MDP5001_342_DPM_Variant_Value_Out_Index_1_REAL_1	:= 		prgEM.stEL3446_IO_1.MDP5001_342_Output.MDP5001_342_DPM_Variant_Value_Out_Index_1_REAL	;
MDP5001_342_DPM_Variant_Value_Out_Index_2_REAL_1	:= 		prgEM.stEL3446_IO_1.MDP5001_342_Output.MDP5001_342_DPM_Variant_Value_Out_Index_2_REAL	;	
MDP5001_342_DPM_Variant_Value_Out_Index_3_REAL_1	:= 		prgEM.stEL3446_IO_1.MDP5001_342_Output.MDP5001_342_DPM_Variant_Value_Out_Index_3_REAL	;
MDP5001_342_DPM_Variant_Value_Out_Index_4_ULINT_1	:= 		prgEM.stEL3446_IO_1.MDP5001_342_Output.MDP5001_342_DPM_Variant_Value_Out_Index_4_ULINT	;
MDP5001_342_DPM_Data_Data_1_1						:= 		prgEM.stEL3446_IO_1.MDP5001_342_Output.MDP5001_342_DPM_Data_Data_1	;
MDP5001_342_DPM_Data_Data_2_1						:= 		prgEM.stEL3446_IO_1.MDP5001_342_Output.MDP5001_342_DPM_Data_Data_2	;
MDP5001_342_DPM_Data_Data_3_1						:= 		prgEM.stEL3446_IO_1.MDP5001_342_Output.MDP5001_342_DPM_Data_Data_3	;
MDP5001_342_DPM_Data_Data_4_1						:= 		prgEM.stEL3446_IO_1.MDP5001_342_Output.MDP5001_342_DPM_Data_Data_4	;
MDP5001_342_DPM_Data_Data_5_1						:= 		prgEM.stEL3446_IO_1.MDP5001_342_Output.MDP5001_342_DPM_Data_Data_5	;
MDP5001_342_DPM_Data_Data_6_1						:= 		prgEM.stEL3446_IO_1.MDP5001_342_Output.MDP5001_342_DPM_Data_Data_6	;
MDP5001_342_DPM_Data_Data_7_1						:= 		prgEM.stEL3446_IO_1.MDP5001_342_Output.MDP5001_342_DPM_Data_Data_7	;
MDP5001_342_DPM_Data_Data_8_1						:= 		prgEM.stEL3446_IO_1.MDP5001_342_Output.MDP5001_342_DPM_Data_Data_8	;
MDP5001_342_DPM_Data_Data_9_1						:= 		prgEM.stEL3446_IO_1.MDP5001_342_Output.MDP5001_342_DPM_Data_Data_9	;
MDP5001_342_DPM_Data_Data_10_1						:= 		prgEM.stEL3446_IO_1.MDP5001_342_Output.MDP5001_342_DPM_Data_Data_10	;
MDP5001_342_DPM_Data_Data_11_1						:= 		prgEM.stEL3446_IO_1.MDP5001_342_Output.MDP5001_342_DPM_Data_Data_11	;
MDP5001_342_DPM_Data_Data_12_1						:= 		prgEM.stEL3446_IO_1.MDP5001_342_Output.MDP5001_342_DPM_Data_Data_12	;
MDP5001_342_DPM_Data_Data_13_1						:= 		prgEM.stEL3446_IO_1.MDP5001_342_Output.MDP5001_342_DPM_Data_Data_13	;
MDP5001_342_DPM_Data_Data_14_1						:= 		prgEM.stEL3446_IO_1.MDP5001_342_Output.MDP5001_342_DPM_Data_Data_14	;
MDP5001_342_DPM_Data_Data_15_1						:= 		prgEM.stEL3446_IO_1.MDP5001_342_Output.MDP5001_342_DPM_Data_Data_15	;
MDP5001_342_DPM_Data_Data_16_1						:= 		prgEM.stEL3446_IO_1.MDP5001_342_Output.MDP5001_342_DPM_Data_Data_16	;
MDP5001_342_DPM_Data_Data_17_1						:= 		prgEM.stEL3446_IO_1.MDP5001_342_Output.MDP5001_342_DPM_Data_Data_17	;
MDP5001_342_DPM_Data_Data_18_1						:= 		prgEM.stEL3446_IO_1.MDP5001_342_Output.MDP5001_342_DPM_Data_Data_18	;
MDP5001_342_DPM_Data_Data_19_1						:= 		prgEM.stEL3446_IO_1.MDP5001_342_Output.MDP5001_342_DPM_Data_Data_19	;
MDP5001_342_DPM_Data_Data_20_1						:= 		prgEM.stEL3446_IO_1.MDP5001_342_Output.MDP5001_342_DPM_Data_Data_20	;




prgEM.stEL3446_IO_2.MDP5001_342_Input.MDP5001_342_I1_Channel_Overcurrent					:=	MDP5001_342_I1_Channel_Overcurrent_2;
prgEM.stEL3446_IO_2.MDP5001_342_Input.MDP5001_342_I1_Channel_Inaccurate_Current			:=	MDP5001_342_I1_Channel_Inaccurate_Current_2;
prgEM.stEL3446_IO_2.MDP5001_342_Input.MDP5001_342_I1_Channel_Current_Guard_Warning		:=	MDP5001_342_I1_Channel_Current_Guard_Warning_2;
prgEM.stEL3446_IO_2.MDP5001_342_Input.MDP5001_342_I1_Channel_Current_Guard_Error			:=	MDP5001_342_I1_Channel_Current_Guard_Error_2;
prgEM.stEL3446_IO_2.MDP5001_342_Input.MDP5001_342_I1_Channel_Apparent_Power_Guard_Warning	:=	MDP5001_342_I1_Channel_Apparent_Power_Guard_Warning_2;
prgEM.stEL3446_IO_2.MDP5001_342_Input.MDP5001_342_I1_Channel_Apparent_Power_Guard_Error	:=	MDP5001_342_I1_Channel_Apparent_Power_Guard_Error_2;
prgEM.stEL3446_IO_2.MDP5001_342_Input.MDP5001_342_I1_Channel_Active_Power_Guard_Warning	:=	MDP5001_342_I1_Channel_Active_Power_Guard_Warning_2;
prgEM.stEL3446_IO_2.MDP5001_342_Input.MDP5001_342_I1_Channel_Active_Power_Guard_Error		:=	MDP5001_342_I1_Channel_Active_Power_Guard_Error_2;
prgEM.stEL3446_IO_2.MDP5001_342_Input.MDP5001_342_I1_Channel_Reactive_Power_Guard_Warning	:=	MDP5001_342_I1_Channel_Reactive_Power_Guard_Warning_2;
prgEM.stEL3446_IO_2.MDP5001_342_Input.MDP5001_342_I1_Channel_Reactive_Power_Guard_Error	:=	MDP5001_342_I1_Channel_Reactive_Power_Guard_Error_2;
prgEM.stEL3446_IO_2.MDP5001_342_Input.MDP5001_342_I1_Channel_DPM_Inaccurate				:=	MDP5001_342_I1_Channel_DPM_Inaccurate_2;
prgEM.stEL3446_IO_2.MDP5001_342_Input.MDP5001_342_I1_Channel_DPM_Timeout					:=	MDP5001_342_I1_Channel_DPM_Timeout_2;
prgEM.stEL3446_IO_2.MDP5001_342_Input.MDP5001_342_I1_Channel_TxPDO_Toggle					:=	MDP5001_342_I1_Channel_TxPDO_Toggle_2;
prgEM.stEL3446_IO_2.MDP5001_342_Input.MDP5001_342_I1_Channel_Current						:=	MDP5001_342_I1_Channel_Current_2;
prgEM.stEL3446_IO_2.MDP5001_342_Input.MDP5001_342_I1_Channel_Active_Power					:=	MDP5001_342_I1_Channel_Active_Power_2;
prgEM.stEL3446_IO_2.MDP5001_342_Input.MDP5001_342_I1_Channel_Apparent_Power				:=	MDP5001_342_I1_Channel_Apparent_Power_2;
prgEM.stEL3446_IO_2.MDP5001_342_Input.MDP5001_342_I1_Channel_Reactive_Power_Fundamental	:=	MDP5001_342_I1_Channel_Reactive_Power_Fundamental_2;
prgEM.stEL3446_IO_2.MDP5001_342_Input.MDP5001_342_I1_Channel_Active_Energy				:=	MDP5001_342_I1_Channel_Active_Energy_2;
prgEM.stEL3446_IO_2.MDP5001_342_Input.MDP5001_342_I2_Channel_Overcurrent					:=	MDP5001_342_I2_Channel_Overcurrent_2;
prgEM.stEL3446_IO_2.MDP5001_342_Input.MDP5001_342_I2_Channel_Inaccurate_Current			:=	MDP5001_342_I2_Channel_Inaccurate_Current_2;
prgEM.stEL3446_IO_2.MDP5001_342_Input.MDP5001_342_I2_Channel_Current_Guard_Warning		:=	MDP5001_342_I2_Channel_Current_Guard_Warning_2;
prgEM.stEL3446_IO_2.MDP5001_342_Input.MDP5001_342_I2_Channel_Current_Guard_Error			:=	MDP5001_342_I2_Channel_Current_Guard_Error_2;
prgEM.stEL3446_IO_2.MDP5001_342_Input.MDP5001_342_I2_Channel_Apparent_Power_Guard_Warning	:=	MDP5001_342_I2_Channel_Apparent_Power_Guard_Warning_2;
prgEM.stEL3446_IO_2.MDP5001_342_Input.MDP5001_342_I2_Channel_Apparent_Power_Guard_Error	:=	MDP5001_342_I2_Channel_Apparent_Power_Guard_Error_2;
prgEM.stEL3446_IO_2.MDP5001_342_Input.MDP5001_342_I2_Channel_Active_Power_Guard_Warning	:=	MDP5001_342_I2_Channel_Active_Power_Guard_Warning_2;
prgEM.stEL3446_IO_2.MDP5001_342_Input.MDP5001_342_I2_Channel_Active_Power_Guard_Error		:=	MDP5001_342_I2_Channel_Active_Power_Guard_Error_2;
prgEM.stEL3446_IO_2.MDP5001_342_Input.MDP5001_342_I2_Channel_Reactive_Power_Guard_Warning	:=	MDP5001_342_I2_Channel_Reactive_Power_Guard_Warning_2;
prgEM.stEL3446_IO_2.MDP5001_342_Input.MDP5001_342_I2_Channel_Reactive_Power_Guard_Error	:=	MDP5001_342_I2_Channel_Reactive_Power_Guard_Error_2;
prgEM.stEL3446_IO_2.MDP5001_342_Input.MDP5001_342_I2_Channel_DPM_Inaccurate				:=	MDP5001_342_I2_Channel_DPM_Inaccurate_2;
prgEM.stEL3446_IO_2.MDP5001_342_Input.MDP5001_342_I2_Channel_DPM_Timeout					:=	MDP5001_342_I2_Channel_DPM_Timeout_2;
prgEM.stEL3446_IO_2.MDP5001_342_Input.MDP5001_342_I2_Channel_TxPDO_Toggle					:=	MDP5001_342_I2_Channel_TxPDO_Toggle_2;
prgEM.stEL3446_IO_2.MDP5001_342_Input.MDP5001_342_I2_Channel_Current						:=	MDP5001_342_I2_Channel_Current_2;
prgEM.stEL3446_IO_2.MDP5001_342_Input.MDP5001_342_I2_Channel_Active_Power					:=	MDP5001_342_I2_Channel_Active_Power_2;
prgEM.stEL3446_IO_2.MDP5001_342_Input.MDP5001_342_I2_Channel_Apparent_Power				:=	MDP5001_342_I2_Channel_Apparent_Power_2;
prgEM.stEL3446_IO_2.MDP5001_342_Input.MDP5001_342_I2_Channel_Reactive_Power_Fundamental	:=	MDP5001_342_I2_Channel_Reactive_Power_Fundamental_2;
prgEM.stEL3446_IO_2.MDP5001_342_Input.MDP5001_342_I2_Channel_Active_Energy				:=	MDP5001_342_I2_Channel_Active_Energy_2;
prgEM.stEL3446_IO_2.MDP5001_342_Input.MDP5001_342_I3_Channel_Overcurrent					:=	MDP5001_342_I3_Channel_Overcurrent_2;
prgEM.stEL3446_IO_2.MDP5001_342_Input.MDP5001_342_I3_Channel_Inaccurate_Current			:=	MDP5001_342_I3_Channel_Inaccurate_Current_2;
prgEM.stEL3446_IO_2.MDP5001_342_Input.MDP5001_342_I3_Channel_Current_Guard_Warning		:=	MDP5001_342_I3_Channel_Current_Guard_Warning_2;
prgEM.stEL3446_IO_2.MDP5001_342_Input.MDP5001_342_I3_Channel_Current_Guard_Error			:=	MDP5001_342_I3_Channel_Current_Guard_Error_2;
prgEM.stEL3446_IO_2.MDP5001_342_Input.MDP5001_342_I3_Channel_Apparent_Power_Guard_Warning	:=	MDP5001_342_I3_Channel_Apparent_Power_Guard_Warning_2;
prgEM.stEL3446_IO_2.MDP5001_342_Input.MDP5001_342_I3_Channel_Apparent_Power_Guard_Error	:=	MDP5001_342_I3_Channel_Apparent_Power_Guard_Error_2;
prgEM.stEL3446_IO_2.MDP5001_342_Input.MDP5001_342_I3_Channel_Active_Power_Guard_Warning	:=	MDP5001_342_I3_Channel_Active_Power_Guard_Warning_2;
prgEM.stEL3446_IO_2.MDP5001_342_Input.MDP5001_342_I3_Channel_Active_Power_Guard_Error		:=	MDP5001_342_I3_Channel_Active_Power_Guard_Error_2;
prgEM.stEL3446_IO_2.MDP5001_342_Input.MDP5001_342_I3_Channel_Reactive_Power_Guard_Warning	:=	MDP5001_342_I3_Channel_Reactive_Power_Guard_Warning_2;
prgEM.stEL3446_IO_2.MDP5001_342_Input.MDP5001_342_I3_Channel_Reactive_Power_Guard_Error	:=	MDP5001_342_I3_Channel_Reactive_Power_Guard_Error_2;
prgEM.stEL3446_IO_2.MDP5001_342_Input.MDP5001_342_I3_Channel_DPM_Inaccurate				:=	MDP5001_342_I3_Channel_DPM_Inaccurate_2;
prgEM.stEL3446_IO_2.MDP5001_342_Input.MDP5001_342_I3_Channel_DPM_Timeout					:=	MDP5001_342_I3_Channel_DPM_Timeout_2;
prgEM.stEL3446_IO_2.MDP5001_342_Input.MDP5001_342_I3_Channel_TxPDO_Toggle					:=	MDP5001_342_I3_Channel_TxPDO_Toggle_2;
prgEM.stEL3446_IO_2.MDP5001_342_Input.MDP5001_342_I3_Channel_Current						:=	MDP5001_342_I3_Channel_Current_2;
prgEM.stEL3446_IO_2.MDP5001_342_Input.MDP5001_342_I3_Channel_Active_Power					:=	MDP5001_342_I3_Channel_Active_Power_2;
prgEM.stEL3446_IO_2.MDP5001_342_Input.MDP5001_342_I3_Channel_Apparent_Power				:=	MDP5001_342_I3_Channel_Apparent_Power_2;
prgEM.stEL3446_IO_2.MDP5001_342_Input.MDP5001_342_I3_Channel_Reactive_Power_Fundamental	:=	MDP5001_342_I3_Channel_Reactive_Power_Fundamental_2;
prgEM.stEL3446_IO_2.MDP5001_342_Input.MDP5001_342_I3_Channel_Active_Energy				:=	MDP5001_342_I3_Channel_Active_Energy_2;
prgEM.stEL3446_IO_2.MDP5001_342_Input.MDP5001_342_I4_Channel_Overcurrent					:=	MDP5001_342_I4_Channel_Overcurrent_2;
prgEM.stEL3446_IO_2.MDP5001_342_Input.MDP5001_342_I4_Channel_Inaccurate_Current			:=	MDP5001_342_I4_Channel_Inaccurate_Current_2;
prgEM.stEL3446_IO_2.MDP5001_342_Input.MDP5001_342_I4_Channel_Current_Guard_Warning		:=	MDP5001_342_I4_Channel_Current_Guard_Warning_2;
prgEM.stEL3446_IO_2.MDP5001_342_Input.MDP5001_342_I4_Channel_Current_Guard_Error			:=	MDP5001_342_I4_Channel_Current_Guard_Error_2;
prgEM.stEL3446_IO_2.MDP5001_342_Input.MDP5001_342_I4_Channel_Apparent_Power_Guard_Warning	:=	MDP5001_342_I4_Channel_Apparent_Power_Guard_Warning_2;
prgEM.stEL3446_IO_2.MDP5001_342_Input.MDP5001_342_I4_Channel_Apparent_Power_Guard_Error	:=	MDP5001_342_I4_Channel_Apparent_Power_Guard_Error_2;
prgEM.stEL3446_IO_2.MDP5001_342_Input.MDP5001_342_I4_Channel_Active_Power_Guard_Warning	:=	MDP5001_342_I4_Channel_Active_Power_Guard_Warning_2;
prgEM.stEL3446_IO_2.MDP5001_342_Input.MDP5001_342_I4_Channel_Active_Power_Guard_Error		:=	MDP5001_342_I4_Channel_Active_Power_Guard_Error_2;
prgEM.stEL3446_IO_2.MDP5001_342_Input.MDP5001_342_I4_Channel_Reactive_Power_Guard_Warning	:=	MDP5001_342_I4_Channel_Reactive_Power_Guard_Warning_2;
prgEM.stEL3446_IO_2.MDP5001_342_Input.MDP5001_342_I4_Channel_Reactive_Power_Guard_Error	:=	MDP5001_342_I4_Channel_Reactive_Power_Guard_Error_2;
prgEM.stEL3446_IO_2.MDP5001_342_Input.MDP5001_342_I4_Channel_DPM_Inaccurate				:=	MDP5001_342_I4_Channel_DPM_Inaccurate_2;
prgEM.stEL3446_IO_2.MDP5001_342_Input.MDP5001_342_I4_Channel_DPM_Timeout					:=	MDP5001_342_I4_Channel_DPM_Timeout_2;
prgEM.stEL3446_IO_2.MDP5001_342_Input.MDP5001_342_I4_Channel_TxPDO_Toggle					:=	MDP5001_342_I4_Channel_TxPDO_Toggle_2;
prgEM.stEL3446_IO_2.MDP5001_342_Input.MDP5001_342_I4_Channel_Current						:=	MDP5001_342_I4_Channel_Current_2;
prgEM.stEL3446_IO_2.MDP5001_342_Input.MDP5001_342_I4_Channel_Active_Power					:=	MDP5001_342_I4_Channel_Active_Power_2;
prgEM.stEL3446_IO_2.MDP5001_342_Input.MDP5001_342_I4_Channel_Apparent_Power				:=	MDP5001_342_I4_Channel_Apparent_Power_2;
prgEM.stEL3446_IO_2.MDP5001_342_Input.MDP5001_342_I4_Channel_Reactive_Power_Fundamental	:=	MDP5001_342_I4_Channel_Reactive_Power_Fundamental_2;
prgEM.stEL3446_IO_2.MDP5001_342_Input.MDP5001_342_I4_Channel_Active_Energy				:=	MDP5001_342_I4_Channel_Active_Energy_2;
prgEM.stEL3446_IO_2.MDP5001_342_Input.MDP5001_342_I5_Channel_Overcurrent					:=	MDP5001_342_I5_Channel_Overcurrent_2;
prgEM.stEL3446_IO_2.MDP5001_342_Input.MDP5001_342_I5_Channel_Inaccurate_Current			:=	MDP5001_342_I5_Channel_Inaccurate_Current_2;
prgEM.stEL3446_IO_2.MDP5001_342_Input.MDP5001_342_I5_Channel_Current_Guard_Warning		:=	MDP5001_342_I5_Channel_Current_Guard_Warning_2;
prgEM.stEL3446_IO_2.MDP5001_342_Input.MDP5001_342_I5_Channel_Current_Guard_Error			:=	MDP5001_342_I5_Channel_Current_Guard_Error_2;
prgEM.stEL3446_IO_2.MDP5001_342_Input.MDP5001_342_I5_Channel_Apparent_Power_Guard_Warning	:=	MDP5001_342_I5_Channel_Apparent_Power_Guard_Warning_2;
prgEM.stEL3446_IO_2.MDP5001_342_Input.MDP5001_342_I5_Channel_Apparent_Power_Guard_Error	:=	MDP5001_342_I5_Channel_Apparent_Power_Guard_Error_2;
prgEM.stEL3446_IO_2.MDP5001_342_Input.MDP5001_342_I5_Channel_Active_Power_Guard_Warning	:=	MDP5001_342_I5_Channel_Active_Power_Guard_Warning_2;
prgEM.stEL3446_IO_2.MDP5001_342_Input.MDP5001_342_I5_Channel_Active_Power_Guard_Error		:=	MDP5001_342_I5_Channel_Active_Power_Guard_Error_2;
prgEM.stEL3446_IO_2.MDP5001_342_Input.MDP5001_342_I5_Channel_Reactive_Power_Guard_Warning	:=	MDP5001_342_I5_Channel_Reactive_Power_Guard_Warning_2;
prgEM.stEL3446_IO_2.MDP5001_342_Input.MDP5001_342_I5_Channel_Reactive_Power_Guard_Error	:=	MDP5001_342_I5_Channel_Reactive_Power_Guard_Error_2;
prgEM.stEL3446_IO_2.MDP5001_342_Input.MDP5001_342_I5_Channel_DPM_Inaccurate				:=	MDP5001_342_I5_Channel_DPM_Inaccurate_2;
prgEM.stEL3446_IO_2.MDP5001_342_Input.MDP5001_342_I5_Channel_DPM_Timeout					:=	MDP5001_342_I5_Channel_DPM_Timeout_2;
prgEM.stEL3446_IO_2.MDP5001_342_Input.MDP5001_342_I5_Channel_TxPDO_Toggle					:=	MDP5001_342_I5_Channel_TxPDO_Toggle_2;
prgEM.stEL3446_IO_2.MDP5001_342_Input.MDP5001_342_I5_Channel_Current						:=	MDP5001_342_I5_Channel_Current_2;
prgEM.stEL3446_IO_2.MDP5001_342_Input.MDP5001_342_I5_Channel_Active_Power					:=	MDP5001_342_I5_Channel_Active_Power_2;
prgEM.stEL3446_IO_2.MDP5001_342_Input.MDP5001_342_I5_Channel_Apparent_Power				:=	MDP5001_342_I5_Channel_Apparent_Power_2;
prgEM.stEL3446_IO_2.MDP5001_342_Input.MDP5001_342_I5_Channel_Reactive_Power_Fundamental	:=	MDP5001_342_I5_Channel_Reactive_Power_Fundamental_2;
prgEM.stEL3446_IO_2.MDP5001_342_Input.MDP5001_342_I5_Channel_Active_Energy				:=	MDP5001_342_I5_Channel_Active_Energy_2;
prgEM.stEL3446_IO_2.MDP5001_342_Input.MDP5001_342_I6_Channel_Overcurrent					:=	MDP5001_342_I6_Channel_Overcurrent_2;
prgEM.stEL3446_IO_2.MDP5001_342_Input.MDP5001_342_I6_Channel_Inaccurate_Current			:=	MDP5001_342_I6_Channel_Inaccurate_Current_2;
prgEM.stEL3446_IO_2.MDP5001_342_Input.MDP5001_342_I6_Channel_Current_Guard_Warning		:=	MDP5001_342_I6_Channel_Current_Guard_Warning_2;
prgEM.stEL3446_IO_2.MDP5001_342_Input.MDP5001_342_I6_Channel_Current_Guard_Error			:=	MDP5001_342_I6_Channel_Current_Guard_Error_2;
prgEM.stEL3446_IO_2.MDP5001_342_Input.MDP5001_342_I6_Channel_Apparent_Power_Guard_Warning	:=	MDP5001_342_I6_Channel_Apparent_Power_Guard_Warning_2;
prgEM.stEL3446_IO_2.MDP5001_342_Input.MDP5001_342_I6_Channel_Apparent_Power_Guard_Error	:=	MDP5001_342_I6_Channel_Apparent_Power_Guard_Error_2;
prgEM.stEL3446_IO_2.MDP5001_342_Input.MDP5001_342_I6_Channel_Active_Power_Guard_Warning	:=	MDP5001_342_I6_Channel_Active_Power_Guard_Warning_2;
prgEM.stEL3446_IO_2.MDP5001_342_Input.MDP5001_342_I6_Channel_Active_Power_Guard_Error		:=	MDP5001_342_I6_Channel_Active_Power_Guard_Error_2;
prgEM.stEL3446_IO_2.MDP5001_342_Input.MDP5001_342_I6_Channel_Reactive_Power_Guard_Warning	:=	MDP5001_342_I6_Channel_Reactive_Power_Guard_Warning_2;
prgEM.stEL3446_IO_2.MDP5001_342_Input.MDP5001_342_I6_Channel_Reactive_Power_Guard_Error	:=	MDP5001_342_I6_Channel_Reactive_Power_Guard_Error_2;
prgEM.stEL3446_IO_2.MDP5001_342_Input.MDP5001_342_I6_Channel_DPM_Inaccurate				:=	MDP5001_342_I6_Channel_DPM_Inaccurate_2;
prgEM.stEL3446_IO_2.MDP5001_342_Input.MDP5001_342_I6_Channel_DPM_Timeout					:=	MDP5001_342_I6_Channel_DPM_Timeout_2;
prgEM.stEL3446_IO_2.MDP5001_342_Input.MDP5001_342_I6_Channel_TxPDO_Toggle					:=	MDP5001_342_I6_Channel_TxPDO_Toggle_2;
prgEM.stEL3446_IO_2.MDP5001_342_Input.MDP5001_342_I6_Channel_Current						:=	MDP5001_342_I6_Channel_Current_2;
prgEM.stEL3446_IO_2.MDP5001_342_Input.MDP5001_342_I6_Channel_Active_Power					:=	MDP5001_342_I6_Channel_Active_Power_2;
prgEM.stEL3446_IO_2.MDP5001_342_Input.MDP5001_342_I6_Channel_Apparent_Power				:=	MDP5001_342_I6_Channel_Apparent_Power_2;
prgEM.stEL3446_IO_2.MDP5001_342_Input.MDP5001_342_I6_Channel_Reactive_Power_Fundamental	:=	MDP5001_342_I6_Channel_Reactive_Power_Fundamental_2;
prgEM.stEL3446_IO_2.MDP5001_342_Input.MDP5001_342_I6_Channel_Active_Energy				:=	MDP5001_342_I6_Channel_Active_Energy_2;
prgEM.stEL3446_IO_2.MDP5001_342_Input.MDP5001_342_DPM_Variant_Value_In_TxPDO_Toggle		:=	MDP5001_342_DPM_Variant_Value_In_TxPDO_Toggle_2;
prgEM.stEL3446_IO_2.MDP5001_342_Input.MDP5001_342_DPM_Variant_Value_In_Index_1_REAL		:=	MDP5001_342_DPM_Variant_Value_In_Index_1_REAL_2;
prgEM.stEL3446_IO_2.MDP5001_342_Input.MDP5001_342_DPM_Variant_Value_In_Value_1_REAL		:=	MDP5001_342_DPM_Variant_Value_In_Value_1_REAL_2;
prgEM.stEL3446_IO_2.MDP5001_342_Input.MDP5001_342_DPM_Variant_Value_In_Index_2_REAL		:=	MDP5001_342_DPM_Variant_Value_In_Index_2_REAL_2;
prgEM.stEL3446_IO_2.MDP5001_342_Input.MDP5001_342_DPM_Variant_Value_In_Value_2_REAL		:=	MDP5001_342_DPM_Variant_Value_In_Value_2_REAL_2;
prgEM.stEL3446_IO_2.MDP5001_342_Input.MDP5001_342_DPM_Variant_Value_In_Index_3_REAL		:=	MDP5001_342_DPM_Variant_Value_In_Index_3_REAL_2;
prgEM.stEL3446_IO_2.MDP5001_342_Input.MDP5001_342_DPM_Variant_Value_In_Value_3_REAL		:=	MDP5001_342_DPM_Variant_Value_In_Value_3_REAL_2;
prgEM.stEL3446_IO_2.MDP5001_342_Input.MDP5001_342_DPM_Variant_Value_In_Index_4_ULINT		:=	MDP5001_342_DPM_Variant_Value_In_Index_4_ULINT_2;
prgEM.stEL3446_IO_2.MDP5001_342_Input.MDP5001_342_DPM_Variant_Value_In_Value_4_ULINT		:=	MDP5001_342_DPM_Variant_Value_In_Value_4_ULINT_2;
       
MDP5001_342_DPM_Variant_Value_Out_Index_1_REAL_2	:= 		prgEM.stEL3446_IO_2.MDP5001_342_Output.MDP5001_342_DPM_Variant_Value_Out_Index_1_REAL	;
MDP5001_342_DPM_Variant_Value_Out_Index_2_REAL_2	:= 		prgEM.stEL3446_IO_2.MDP5001_342_Output.MDP5001_342_DPM_Variant_Value_Out_Index_2_REAL	;	
MDP5001_342_DPM_Variant_Value_Out_Index_3_REAL_2	:= 		prgEM.stEL3446_IO_2.MDP5001_342_Output.MDP5001_342_DPM_Variant_Value_Out_Index_3_REAL	;
MDP5001_342_DPM_Variant_Value_Out_Index_4_ULINT_2	:= 		prgEM.stEL3446_IO_2.MDP5001_342_Output.MDP5001_342_DPM_Variant_Value_Out_Index_4_ULINT	;
MDP5001_342_DPM_Data_Data_1_2						:= 		prgEM.stEL3446_IO_2.MDP5001_342_Output.MDP5001_342_DPM_Data_Data_1	;
MDP5001_342_DPM_Data_Data_2_2						:= 		prgEM.stEL3446_IO_2.MDP5001_342_Output.MDP5001_342_DPM_Data_Data_2	;
MDP5001_342_DPM_Data_Data_3_2						:= 		prgEM.stEL3446_IO_2.MDP5001_342_Output.MDP5001_342_DPM_Data_Data_3	;
MDP5001_342_DPM_Data_Data_4_2						:= 		prgEM.stEL3446_IO_2.MDP5001_342_Output.MDP5001_342_DPM_Data_Data_4	;
MDP5001_342_DPM_Data_Data_5_2						:= 		prgEM.stEL3446_IO_2.MDP5001_342_Output.MDP5001_342_DPM_Data_Data_5	;
MDP5001_342_DPM_Data_Data_6_2						:= 		prgEM.stEL3446_IO_2.MDP5001_342_Output.MDP5001_342_DPM_Data_Data_6	;
MDP5001_342_DPM_Data_Data_7_2						:= 		prgEM.stEL3446_IO_2.MDP5001_342_Output.MDP5001_342_DPM_Data_Data_7	;
MDP5001_342_DPM_Data_Data_8_2						:= 		prgEM.stEL3446_IO_2.MDP5001_342_Output.MDP5001_342_DPM_Data_Data_8	;
MDP5001_342_DPM_Data_Data_9_2						:= 		prgEM.stEL3446_IO_2.MDP5001_342_Output.MDP5001_342_DPM_Data_Data_9	;
MDP5001_342_DPM_Data_Data_10_2						:= 		prgEM.stEL3446_IO_2.MDP5001_342_Output.MDP5001_342_DPM_Data_Data_10	;
MDP5001_342_DPM_Data_Data_11_2						:= 		prgEM.stEL3446_IO_2.MDP5001_342_Output.MDP5001_342_DPM_Data_Data_11	;
MDP5001_342_DPM_Data_Data_12_2						:= 		prgEM.stEL3446_IO_2.MDP5001_342_Output.MDP5001_342_DPM_Data_Data_12	;
MDP5001_342_DPM_Data_Data_13_2						:= 		prgEM.stEL3446_IO_2.MDP5001_342_Output.MDP5001_342_DPM_Data_Data_13	;
MDP5001_342_DPM_Data_Data_14_2						:= 		prgEM.stEL3446_IO_2.MDP5001_342_Output.MDP5001_342_DPM_Data_Data_14	;
MDP5001_342_DPM_Data_Data_15_2						:= 		prgEM.stEL3446_IO_2.MDP5001_342_Output.MDP5001_342_DPM_Data_Data_15	;
MDP5001_342_DPM_Data_Data_16_2						:= 		prgEM.stEL3446_IO_2.MDP5001_342_Output.MDP5001_342_DPM_Data_Data_16	;
MDP5001_342_DPM_Data_Data_17_2						:= 		prgEM.stEL3446_IO_2.MDP5001_342_Output.MDP5001_342_DPM_Data_Data_17	;
MDP5001_342_DPM_Data_Data_18_2						:= 		prgEM.stEL3446_IO_2.MDP5001_342_Output.MDP5001_342_DPM_Data_Data_18	;
MDP5001_342_DPM_Data_Data_19_2						:= 		prgEM.stEL3446_IO_2.MDP5001_342_Output.MDP5001_342_DPM_Data_Data_19	;
MDP5001_342_DPM_Data_Data_20_2						:= 		prgEM.stEL3446_IO_2.MDP5001_342_Output.MDP5001_342_DPM_Data_Data_20	;

END_PROGRAM

(* stored: Version 1.1.0.1, ProductVersion 3.1.4024.12
   POU prgHW: Id {fb8718a3-389b-4d9b-b3ed-ea76bac0641c}, SpecialFunc None *)
